(* CODESYS project FBD_TON.project

Project tree, tasks and I/O mapping:
  Device : CODESYS Control Win V3, 3S - Smart Software Solutions GmbH, version 3.5.15.30
    application Application
      libraries: Standard, * (System)
      task MainTask (cyclic, interval t#20ms, priority 1) calls PLC_PRG
      task VISU_TASK (cyclic, interval 100 ms, priority 31) calls VisuElems.Visu_Prg
      program PLC_PRG [FBD]
      visualisation Visualization
  text list GlobalTextList
*)

// Device/Application/PLC_PRG
PROGRAM PLC_PRG
VAR
	TON_0: TON;
	TON_0_IN: BOOL;
	TON_0_PT: TIME := T#5s;
	TON_0_ET: TIME;
	TON_0_Q: BOOL;
END_VAR

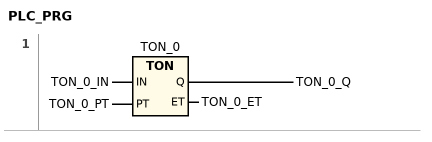
// NETWORK 1
TON_0(IN := TON_0_IN, PT := TON_0_PT, ET => TON_0_ET); // TON
TON_0_Q := TON_0.Q;

END_PROGRAM

// Device/Application/Visualization
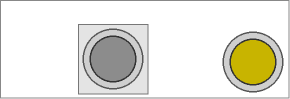
VISUALIZATION Visualization  // 290x99
    Lamp1 (218,27 70x70), variable: PLC_PRG.TON_0_Q, style: Lamp-Lamp1-Yellow
    PushSwitch (78,24 70x70), variable: PLC_PRG.TON_0_IN, behaviour: TOGGLE, style: Switch-PushSwitch-Gray
END_VISUALIZATION
